ABB RobotStudio station: IRB120 Polishing.rsstn

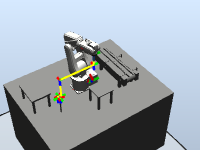
Station Solution5 (saved by RobotStudio 6.8.8148.134)
Controller System1, task T_ROB1: task frame (RAPID world) sits at (0, 9.13, 947.51) mm, rotated rx 0 ry 0 rz 180 deg in the station
Controller System1
  mechanical unit ROB_1: IRB120_3_58__01, 6 joints, base frame (-22.73, 0, 0) mm
Layout (positions relative to the parent item):
  - 零件1 [part] at (0, 0, 514.4) mm, rotated rx 90 ry 0 rz 0 deg
  - IRB120_3_58__01 [mechanism] at (22.73, 9.13, 947.51) mm, rotated rx 0 ry 0 rz 180 deg; joint values [1.803, -0.306, 0.1892, 0, 1.6876, 0.2322] (rad or m)
      links: Base, Link1, Link2, Link3, Link4, Link5, Link6
  - 部件_2 [part] at (71.17, -195.66, 1527.69) mm, rotated rx 180 ry 0 rz 90 deg
  - 部件_5 [part] at (-353.84, -202.68, 942.84) mm
  - 部件_7 [part] at (-349.68, -195.66, 1086.83) mm
  - 写字台 [part] at (-601.17, 227.59, 1145.08) mm, rotated rx 90 ry 0 rz 0 deg
Attachment: 部件_2 is attached to IRB120_3_58__01 / Link6
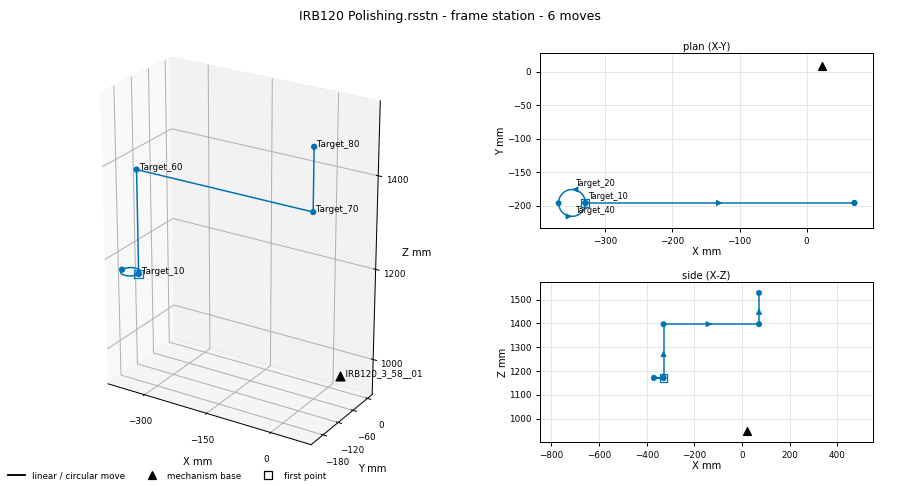
[picture p0: tool path of IRB120 Polishing.rsstn in frame station, 6 of 6 moves have a stored position in this frame; points joined in program order, loops and branches not executed]
Targets, tools, work objects and paths stored in the station, written as RAPID:
! task T_ROB1
MODULE CalibData
  PERS tooldata Weldgun:=[TRUE,[[20.31,0,363.689],[0.948464781,0,0.316882565,0]],[1,[0,0,1],[1,0,0,0],0,0,0]];
  PERS tooldata ROBOBEL926_T_TD_0:=[TRUE,[[117,0,470],[0.866025404,0,0.5,0]],[5.5,[30,0,225],[1,0,0,0],0,0,0]];
  PERS tooldata ROBOBEL926_T_TD_100:=[TRUE,[[204,0,520],[0.866025404,0,0.5,0]],[5.5,[30,0,225],[1,0,0,0],0,0,0]];
  PERS tooldata ROBOBEL926_T_TD_120:=[TRUE,[[220,0,530],[0.866025404,0,0.5,0]],[5.5,[30,0,225],[1,0,0,0],0,0,0]];
  PERS tooldata ROBOBEL926_T_TD_150:=[TRUE,[[247,0,545],[0.866025404,0,0.5,0]],[5.5,[30,0,225],[1,0,0,0],0,0,0]];
  PERS tooldata ROBOBEL926_T_TD_200:=[TRUE,[[290,0,570],[0.866025404,0,0.5,0]],[5.5,[30,0,225],[1,0,0,0],0,0,0]];
  PERS tooldata ROBOBEL926_T_TD_250:=[TRUE,[[333,0,595],[0.866025404,0,0.5,0]],[5.5,[30,0,225],[1,0,0,0],0,0,0]];
  PERS tooldata ROBOBEL926_T_TD_300:=[TRUE,[[377,0,620],[0.866025404,0,0.5,0]],[5.5,[30,0,225],[1,0,0,0],0,0,0]];
ENDMODULE

! task T_ROB1
MODULE Module1
  CONST robtarget Target_10:=[[329.684821514,204.795803999,223.736626115],[0,-0.707106781,0.707106781,0],[0,0,0,0],[9E+09,9E+09,9E+09,9E+09,9E+09,9E+09]];
  CONST robtarget Target_20:=[[349.907624895,184.797045072,223.736626115],[0,0.999984486,0.005570171,0],[0,0,-2,0],[9E+09,9E+09,9E+09,9E+09,9E+09,9E+09]];
  CONST robtarget Target_30:=[[369.679857379,205.24138311,223.736626115],[0,0.699185614,0.714940192,0],[0,0,-3,0],[9E+09,9E+09,9E+09,9E+09,9E+09,9E+09]];
  CONST robtarget Target_40:=[[349.462018133,224.794562927,223.736626115],[0,-0.005570171,0.999984486,0],[0,0,-4,0],[9E+09,9E+09,9E+09,9E+09,9E+09,9E+09]];
  CONST robtarget Target_50:=[[329.684821514,204.795803999,223.736626115],[0,-0.707106781,0.707106781,0],[0,0,0,0],[9E+09,9E+09,9E+09,9E+09,9E+09,9E+09]];
  CONST robtarget Target_60:=[[329.684769595,204.795804402,449.106771309],[-0.000000025,0.707106797,-0.707106766,-0.000000007],[0,0,-1,0],[9E+09,9E+09,9E+09,9E+09,9E+09,9E+09]];
  CONST robtarget Target_70:=[[-71.165455598,204.795809158,449.106776254],[0.000000011,-0.707106764,0.707106799,0.000000015],[1,-1,0,0],[9E+09,9E+09,9E+09,9E+09,9E+09,9E+09]];
  CONST robtarget Target_80:=[[-71.165454684,204.795805292,580.184186337],[-0.000000004,-0.707106779,0.707106783,0.000000041],[1,0,0,0],[9E+09,9E+09,9E+09,9E+09,9E+09,9E+09]];
  PROC Path_10()
    MoveL Target_10,v100,fine,tool0\WObj:=wobj0;
    MoveC Target_20,Target_30,v100,fine,tool0\WObj:=wobj0;
    MoveC Target_40,Target_50,v100,fine,tool0\WObj:=wobj0;
    MoveL Target_60,v100,fine,tool0\WObj:=wobj0;
    MoveL Target_70,v100,fine,tool0\WObj:=wobj0;
    MoveL Target_80,v100,fine,tool0\WObj:=wobj0;
  ENDPROC
  PROC main()
  ENDPROC
ENDMODULE

